FUNCTION_BLOCK hsv2rgb (* Simple helper function, converting HSV color space to RGB color space *)
  (* Standard: 61499-2; Description: Copyright (c) 2022 HR Agrartechnik GmbH This program and the accompanying materials are made available under the terms of the Eclipse Public License 2.0 which is available at https://www.eclipse.org/legal/epl-2.0/ SPDX-License-Identifier: EPL-2.0 Wiki: https://en.wikipedia.org/wiki/HSL_and_HSV *)
  (* Version 1.0, 2022-07-16, Franz Höpfinger, HR Agrartechnik GmbH *)
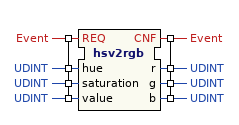
  EVENT_INPUT
    REQ WITH hue, saturation, value; (* Service Request *)
  END_EVENT
  EVENT_OUTPUT
    CNF WITH r, g, b; (* Confirmation of Requested Service *)
  END_EVENT
  VAR_INPUT
    hue : UDINT; (* hue *)
    saturation : UDINT; (* saturation *)
    value : UDINT; (* value *)
  END_VAR
  VAR_OUTPUT
    r : UDINT; (* red *)
    g : UDINT; (* green *)
    b : UDINT; (* blue *)
  END_VAR
END_FUNCTION_BLOCK
